{attribute 'qualified_only'}
VAR_GLOBAL
	
	rosData : ST_hyflowROS;

END_VAR

(* stored: Version 1.1.0.1
   GVL GVL_HyFlow: Id {d0d666e7-02f6-4dfd-a8e0-2097e2940ae1} *)
